FUNCTION_BLOCK xPPU_LSC
VAR_INPUT
	i_error: POINTER TO ErrorManager;
	i_process: POINTER TO ProcessManager;
	i_state: POINTER TO StateTracker;
END_VAR
VAR
	m_conveyorParams: ParameterSet;
	m_subRes: EOperationResult;
END_VAR

VAR
	m_alarm_flags: ARRAY [1..10] OF BOOL := [FALSE, FALSE, FALSE, FALSE, FALSE, FALSE,FALSE, FALSE, FALSE, FALSE];
	m_timer_LSC_WPStartCheck : TON;
	
	m_timer_LSC_SwitchRetracted: TON;
	LSC_MetalWPAtStart_History : BOOL := FALSE; 
    LSC_MetalWPAtMid_History : BOOL := FALSE;
	LSC_LightWPAtStart_History: BOOL:= FALSE;
	LSC_LightWPAtMid_History: BOOL:= FALSE;
	LSC_LightWPAtEnd_History: BOOL:= FALSE;
END_VAR

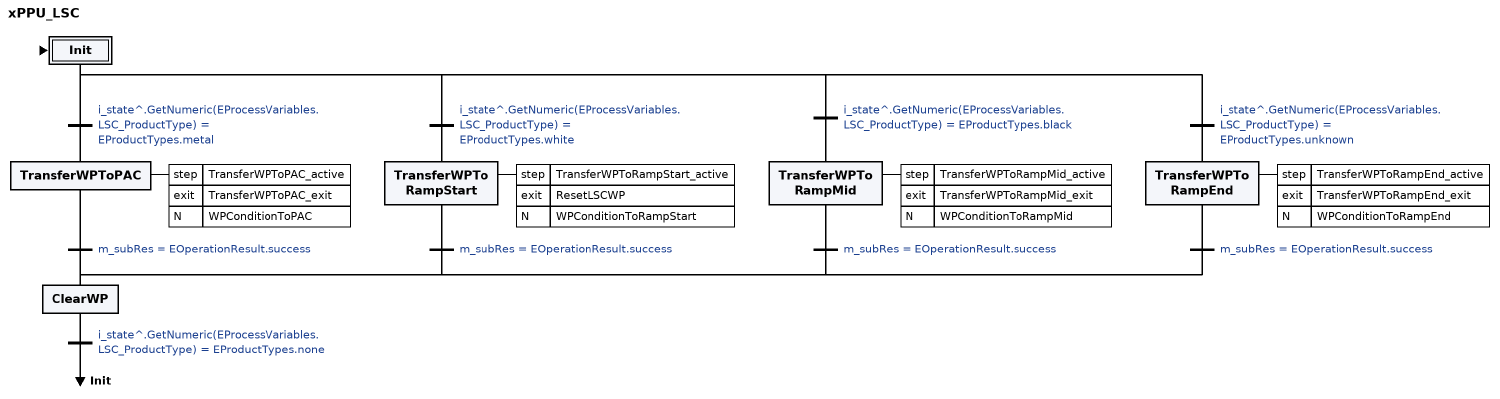
INITIAL_STEP Init:
END_STEP
TRANSITION FROM Init TO TransferWPToPAC
    := i_state^.GetNumeric(EProcessVariables.LSC_ProductType) = EProductTypes.metal;
END_TRANSITION
STEP TransferWPToPAC:
    TransferWPToPAC_active(N);  // step action
    TransferWPToPAC_exit(P0);  // exit action
    WPConditionToPAC(N);
END_STEP
TRANSITION FROM TransferWPToPAC TO ClearWP
    := m_subRes = EOperationResult.success;
END_TRANSITION
TRANSITION FROM Init TO TransferWPToRampStart
    := i_state^.GetNumeric(EProcessVariables.LSC_ProductType) = EProductTypes.white;
END_TRANSITION
STEP TransferWPToRampStart:
    TransferWPToRampStart_active(N);  // step action
    ResetLSCWP(P0);  // exit action
    WPConditionToRampStart(N);
END_STEP
TRANSITION FROM TransferWPToRampStart TO ClearWP
    := m_subRes = EOperationResult.success;
END_TRANSITION
TRANSITION FROM Init TO TransferWPToRampMid
    := i_state^.GetNumeric(EProcessVariables.LSC_ProductType) = EProductTypes.black;
END_TRANSITION
STEP TransferWPToRampMid:
    TransferWPToRampMid_active(N);  // step action
    TransferWPToRampMid_exit(P0);  // exit action
    WPConditionToRampMid(N);
END_STEP
TRANSITION FROM TransferWPToRampMid TO ClearWP
    := m_subRes = EOperationResult.success;
END_TRANSITION
TRANSITION FROM Init TO TransferWPToRampEnd
    := i_state^.GetNumeric(EProcessVariables.LSC_ProductType) = EProductTypes.unknown;
END_TRANSITION
STEP TransferWPToRampEnd:
    TransferWPToRampEnd_active(N);  // step action
    TransferWPToRampEnd_exit(P0);  // exit action
    WPConditionToRampEnd(N);
END_STEP
TRANSITION FROM TransferWPToRampEnd TO ClearWP
    := m_subRes = EOperationResult.success;
END_TRANSITION
STEP ClearWP:
END_STEP
TRANSITION FROM ClearWP TO Init
    := i_state^.GetNumeric(EProcessVariables.LSC_ProductType) = EProductTypes.none;
END_TRANSITION

ACTION ResetLSCWP:
i_state^.ShiftProduct(EProducts.LSC_product,0);
END_ACTION

ACTION TransferWPAtStart_active:
m_subRes := i_process^.Execute(
	EBehaviorType.control_primitive,
	EPrimitives.LSC_TransferWPAtStart,
	m_conveyorParams);
END_ACTION

ACTION TransferWPToPAC_active:
m_subRes := i_process^.Execute(
	EBehaviorType.control_primitive,
	EPrimitives.LSC_TransferWorkpieceTo_PAC,
	m_conveyorParams);
	
IF i_state^.GetBinary(EProcessVariables.LSC_LightWPAtStart) THEN
    LSC_LightWPAtStart_History := TRUE;
END_IF

IF i_state^.GetBinary(EProcessVariables.LSC_LightWPAtStart) THEN
    LSC_LightWPAtMid_History := TRUE;
END_IF

IF i_state^.GetBinary(EProcessVariables.LSC_LightWPAtEnd) THEN
    LSC_LightWPAtEnd_History := TRUE;
END_IF

IF i_state^.GetBinary(EProcessVariables.LSC_MetalWPAtStart) THEN
    LSC_MetalWPAtStart_History := TRUE;
END_IF

IF i_state^.GetBinary(EProcessVariables.LSC_MetalWPAtMid) THEN
    LSC_MetalWPAtMid_History := TRUE;
END_IF
END_ACTION

ACTION TransferWPToPAC_exit:
i_state^.ShiftProduct(EProducts.LSC_product,0);

IF m_alarm_flags[2]= FALSE 
	AND (NOT LSC_MetalWPAtStart_History) //OR NOT LSC_MetalWPAtMid_History)
	OR (NOT LSC_LightWPAtMid_History OR NOT LSC_MetalWPAtMid_History)
	OR LSC_LightWPAtEnd_History
THEN
    i_error^.AddMessage(EAlarms.LSC_WPType_ToPAC_changed, TRUE, ESeverity.error, 'WPType on LSC changed from Metal to others');
	m_alarm_flags[2] := TRUE;
END_IF
LSC_MetalWPAtStart_History := FALSE;
LSC_MetalWPAtMid_History := FALSE;
END_ACTION

ACTION TransferWPToRampEnd_active:
m_subRes := i_process^.Execute(
	EBehaviorType.control_primitive,
	EPrimitives.LSC_TransferWorkpieceTo_RampEnd,
	m_conveyorParams);

IF i_state^.GetBinary(EProcessVariables.LSC_LightWPAtStart) THEN
    LSC_LightWPAtStart_History := TRUE;
END_IF

IF i_state^.GetBinary(EProcessVariables.LSC_LightWPAtStart) THEN
    LSC_LightWPAtMid_History := TRUE;
END_IF

IF i_state^.GetBinary(EProcessVariables.LSC_LightWPAtEnd) THEN
    LSC_LightWPAtEnd_History := TRUE;
END_IF

IF i_state^.GetBinary(EProcessVariables.LSC_MetalWPAtStart) THEN
    LSC_MetalWPAtStart_History := TRUE;
END_IF

IF i_state^.GetBinary(EProcessVariables.LSC_MetalWPAtMid) THEN
    LSC_MetalWPAtMid_History := TRUE;
END_IF
END_ACTION

ACTION TransferWPToRampEnd_exit:
i_state^.ShiftProduct(EProducts.LSC_product,0);

IF m_alarm_flags[5]= FALSE 
	AND (LSC_LightWPAtStart_History) //OR NOT LSC_MetalWPAtStart_History)
	OR (LSC_LightWPAtMid_History OR NOT LSC_MetalWPAtMid_History)
	OR LSC_LightWPAtEnd_History
THEN
    i_error^.AddMessage(EAlarms.LSC_WPType_ToRampEnd_changed, TRUE, ESeverity.error, 'WPType on LSC changed from unknown to others');
	m_alarm_flags[5] := TRUE;
END_IF

LSC_LightWPAtStart_History := FALSE;
LSC_LightWPAtMid_History := FALSE;
LSC_LightWPAtEnd_History := FALSE;
LSC_MetalWPAtStart_History := FALSE;
LSC_MetalWPAtMid_History := FALSE;
END_ACTION

ACTION TransferWPToRampMid_active:
m_subRes := i_process^.Execute(
	EBehaviorType.control_primitive,
	EPrimitives.LSC_TransferWorkpieceTo_RampMid,
	m_conveyorParams);

IF i_state^.GetBinary(EProcessVariables.LSC_LightWPAtStart) THEN
    LSC_LightWPAtStart_History := TRUE;
END_IF

IF i_state^.GetBinary(EProcessVariables.LSC_LightWPAtStart) THEN
    LSC_LightWPAtMid_History := TRUE;
END_IF

IF i_state^.GetBinary(EProcessVariables.LSC_LightWPAtEnd) THEN
    LSC_LightWPAtEnd_History := TRUE;
END_IF

IF i_state^.GetBinary(EProcessVariables.LSC_MetalWPAtStart) THEN
    LSC_MetalWPAtStart_History := TRUE;
END_IF

IF i_state^.GetBinary(EProcessVariables.LSC_MetalWPAtMid) THEN
    LSC_MetalWPAtMid_History := TRUE;
END_IF
END_ACTION

ACTION TransferWPToRampMid_exit:
i_state^.ShiftProduct(EProducts.LSC_product,0);

IF m_alarm_flags[4]= FALSE 
	AND (LSC_LightWPAtStart_History) //OR LSC_LightWPAtMid_History)
	OR (LSC_LightWPAtMid_History OR LSC_MetalWPAtMid_History)
	OR LSC_LightWPAtEnd_History
THEN
    i_error^.AddMessage(EAlarms.LSC_WPType_ToRampMid_changed, TRUE, ESeverity.error, 'WPType on LSC changed from Black to others');
	m_alarm_flags[4] := TRUE;
END_IF
LSC_LightWPAtStart_History := FALSE;
LSC_LightWPAtMid_History := FALSE;
END_ACTION

ACTION TransferWPToRampStart_active:
m_subRes := i_process^.Execute(
	EBehaviorType.control_primitive,
	EPrimitives.LSC_TransferWorkpieceTo_RampStart,
	m_conveyorParams);

IF i_state^.GetBinary(EProcessVariables.LSC_LightWPAtStart) THEN
    LSC_LightWPAtStart_History := TRUE;
END_IF

IF i_state^.GetBinary(EProcessVariables.LSC_LightWPAtStart) THEN
    LSC_LightWPAtMid_History := TRUE;
END_IF

IF i_state^.GetBinary(EProcessVariables.LSC_LightWPAtEnd) THEN
    LSC_LightWPAtEnd_History := TRUE;
END_IF

IF i_state^.GetBinary(EProcessVariables.LSC_MetalWPAtStart) THEN
    LSC_MetalWPAtStart_History := TRUE;
END_IF

IF i_state^.GetBinary(EProcessVariables.LSC_MetalWPAtMid) THEN
    LSC_MetalWPAtMid_History := TRUE;
END_IF
END_ACTION

ACTION TransferWPToRampStart_exit:
//i_state^.ShiftProduct(EProducts.LSC_product,0);

IF m_alarm_flags[3]= FALSE 
	AND (NOT LSC_LightWPAtStart_History) //OR LSC_MetalWPAtStart_History)
	OR (LSC_LightWPAtMid_History OR LSC_MetalWPAtMid_History 
	OR LSC_LightWPAtEnd_History)
THEN
    i_error^.AddMessage(EAlarms.LSC_WPType_ToRampStart_changed, TRUE, ESeverity.error, 'WPType on LSC changed from White to others');
	m_alarm_flags[3] := TRUE;
END_IF
LSC_LightWPAtStart_History := FALSE;
END_ACTION

ACTION WPConditionToPAC:
IF (i_state^.GetNumeric(EProcessVariables.LSC_ProductType) > 0) THEN
    m_timer_LSC_WPStartCheck(IN := TRUE, PT := T#3000MS);
ELSE
    m_timer_LSC_WPStartCheck(IN := FALSE); 
END_IF

IF i_state^.GetBinary(EProcessVariables.LSC_WorkpieceAtEntry) THEN
    m_timer_LSC_WPStartCheck(IN := FALSE);
END_IF

IF m_alarm_flags[1] = FALSE
   AND m_timer_LSC_WPStartCheck.Q 
THEN
    i_error^.AddMessage(EAlarms.LSC_WP_abnormal_Entry, TRUE, ESeverity.error, 'WP not corrctly pass by the Presence sensor at Entry of LSC');
    m_alarm_flags[1] := TRUE; 
END_IF
END_ACTION

ACTION WPConditionToRampEnd:
IF (i_state^.GetNumeric(EProcessVariables.LSC_ProductType) > 0) THEN
    m_timer_LSC_WPStartCheck(IN := TRUE, PT := T#5000MS);
ELSE
    m_timer_LSC_WPStartCheck(IN := FALSE); 
END_IF;

IF i_state^.GetBinary(EProcessVariables.LSC_WorkpieceAtEntry) THEN
    m_timer_LSC_WPStartCheck(IN := FALSE);
END_IF;

IF m_alarm_flags[1] = FALSE
   AND m_timer_LSC_WPStartCheck.Q 
THEN
    i_error^.AddMessage(EAlarms.LSC_WP_abnormal_Entry, TRUE, ESeverity.error, 'WP not correctly pass by the Presence sensor at Entry of LSC');
    m_alarm_flags[1] := TRUE; 
END_IF;
END_ACTION

ACTION WPConditionToRampMid:
IF (i_state^.GetNumeric(EProcessVariables.LSC_ProductType) > 0) THEN
    m_timer_LSC_WPStartCheck(IN := TRUE, PT := T#5000MS);
ELSE
    m_timer_LSC_WPStartCheck(IN := FALSE); 
END_IF;

IF i_state^.GetBinary(EProcessVariables.LSC_WorkpieceAtEntry) THEN
    m_timer_LSC_WPStartCheck(IN := FALSE);
END_IF;

IF m_alarm_flags[1] = FALSE
   AND m_timer_LSC_WPStartCheck.Q 
THEN
    i_error^.AddMessage(EAlarms.LSC_WP_abnormal_Entry, TRUE, ESeverity.error, 'WP not correctly pass by the Presence sensor at Entry of LSC');
    m_alarm_flags[1] := TRUE; 
END_IF;
END_ACTION

ACTION WPConditionToRampStart:
IF (i_state^.GetNumeric(EProcessVariables.LSC_ProductType) > 0) THEN
    m_timer_LSC_WPStartCheck(IN := TRUE, PT := T#4000MS);
ELSE
    m_timer_LSC_WPStartCheck(IN := FALSE); 
END_IF;

IF i_state^.GetBinary(EProcessVariables.LSC_WorkpieceAtEntry) THEN
    m_timer_LSC_WPStartCheck(IN := FALSE);
END_IF;

IF m_alarm_flags[1] = FALSE
   AND m_timer_LSC_WPStartCheck.Q 
THEN
    i_error^.AddMessage(EAlarms.LSC_WP_abnormal_Entry, TRUE, ESeverity.error, 'WP not correctly pass by the Presence sensor at Entry of LSC');
    m_alarm_flags[1] := TRUE; 
END_IF;
END_ACTION

END_FUNCTION_BLOCK

(* stored: Version 1.1.0.1
   POU xPPU_LSC: Id {8246a5de-9303-4982-9c16-a709139cb910}, SpecialFunc None
   Action ResetLSCWP: Id {7fb1714f-6424-4786-a5e1-3c86619d5b06}
   Action TransferWPAtStart_active: Id {17568f3d-2c6e-49c8-8ccd-3fd63d5a5f11}
   Action TransferWPToPAC_active: Id {52233bd1-b3db-4254-98fc-82373ff14cb5}
   Action TransferWPToPAC_exit: Id {c6d5580b-50cd-4045-abcf-5927562f5abb}
   Action TransferWPToRampEnd_active: Id {e1536d26-ab26-4cec-8e9e-336f227510b4}
   Action TransferWPToRampEnd_exit: Id {40ded3d1-e241-44f1-845b-8dbc8e186101}
   Action TransferWPToRampMid_active: Id {4bd98ecb-0488-416f-a2ed-b9eddd1c18f1}
   Action TransferWPToRampMid_exit: Id {f73ccbdb-5c30-473d-98a7-0dcc82be94d1}
   Action TransferWPToRampStart_active: Id {cec12bdf-7a2b-4fd0-8f98-bc04b09d656d}
   Action TransferWPToRampStart_exit: Id {08571f07-2132-4ee2-ab91-9732ae3ba43a}
   Action WPConditionToPAC: Id {b920f8b9-1ebd-4d15-a6f7-dc905b88b8ac}
   Action WPConditionToRampEnd: Id {6e21f871-876c-49f1-8383-0210929b4420}
   Action WPConditionToRampMid: Id {c16c0323-d2d3-4980-a9c1-8904bb67f25e}
   Action WPConditionToRampStart: Id {1e84d262-406b-4a28-b0ea-bdb4aa66402c} *)
